PROGRAM F15_ClusterCtrl_Larm
VAR
	tof_0: TOF;

	FB_FL0: FB_FL;
	FB_FL1: FB_FL;
	FB_FL2: FB_FL;
	FB_FL3: FB_FL;
	FB_FL4: FB_FL;
	FB_FL5: FB_FL;
	FB_FL6: FB_FL;
	test: INT;
END_VAR
VAR // added by the converter: edge detectors and wires of the graphical bodies
    _w1, _w2 : ANY;
END_VAR

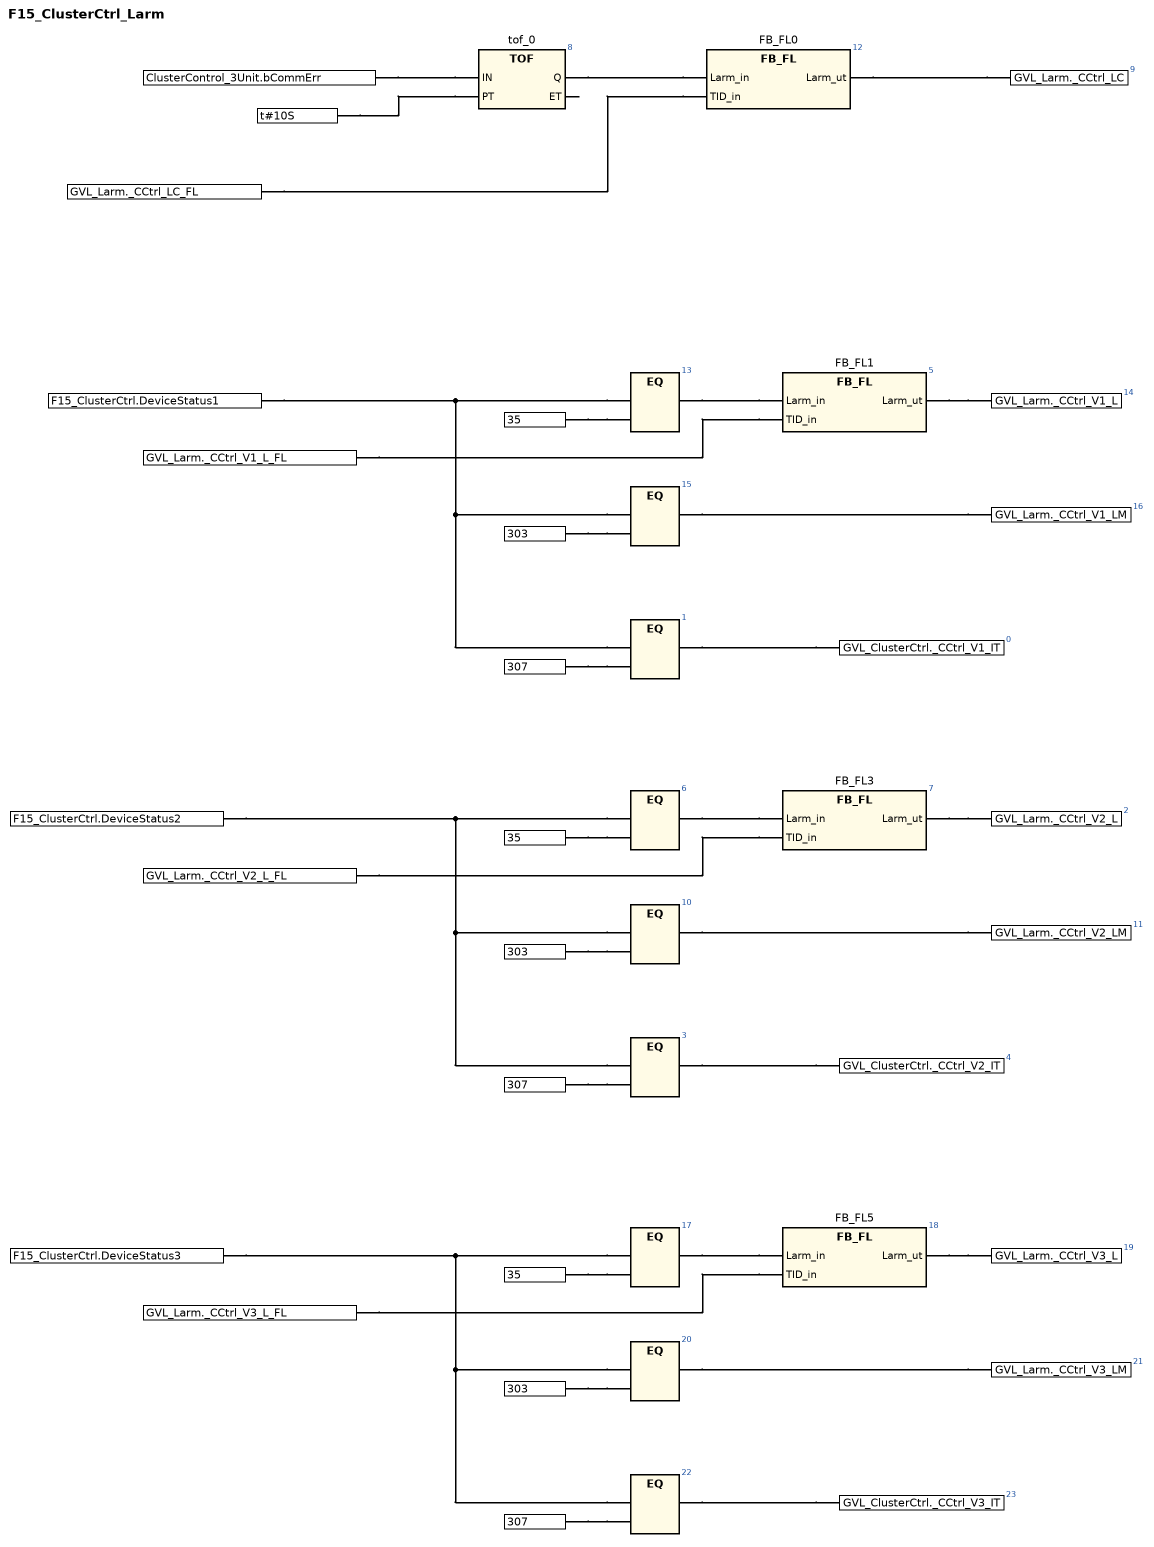
GVL_ClusterCtrl._CCtrl_V1_IT := _w1;
_w1 := F15_ClusterCtrl.DeviceStatus1 = 307;
GVL_Larm._CCtrl_V2_L := FB_FL3.Larm_ut;
GVL_ClusterCtrl._CCtrl_V2_IT := F15_ClusterCtrl.DeviceStatus2 = 307;
FB_FL1(Larm_in := _w2, TID_in := GVL_Larm._CCtrl_V1_L_FL); // FB_FL
FB_FL3(Larm_in := F15_ClusterCtrl.DeviceStatus2 = 35, TID_in := GVL_Larm._CCtrl_V2_L_FL); // FB_FL
tof_0(IN := ClusterControl_3Unit.bCommErr, PT := t#10S); // TOF
GVL_Larm._CCtrl_LC := FB_FL0.Larm_ut;
GVL_Larm._CCtrl_V2_LM := F15_ClusterCtrl.DeviceStatus2 = 303;
FB_FL0(Larm_in := tof_0.Q, TID_in := GVL_Larm._CCtrl_LC_FL); // FB_FL
_w2 := F15_ClusterCtrl.DeviceStatus1 = 35;
GVL_Larm._CCtrl_V1_L := FB_FL1.Larm_ut;
GVL_Larm._CCtrl_V1_LM := F15_ClusterCtrl.DeviceStatus1 = 303;
FB_FL5(Larm_in := F15_ClusterCtrl.DeviceStatus3 = 35, TID_in := GVL_Larm._CCtrl_V3_L_FL); // FB_FL
GVL_Larm._CCtrl_V3_L := FB_FL5.Larm_ut;
GVL_Larm._CCtrl_V3_LM := F15_ClusterCtrl.DeviceStatus3 = 303;
GVL_ClusterCtrl._CCtrl_V3_IT := F15_ClusterCtrl.DeviceStatus3 = 307;

END_PROGRAM

(* stored: Version 1.1.0.1, ProductVersion 3.1.4020.12
   POU F15_ClusterCtrl_Larm: Id {6821dc94-73cd-4723-92e9-4d9cc55bb4d4}, SpecialFunc None *)
